{attribute 'qualified_only'}
{attribute 'strict'}
{attribute 'to_string'}
TYPE E_GridTypeSelection :
(
  Default             := 0,  // Default deformation based on cam points
  None                := 1,  // No deformation calculated all dx/dy=0
  Test_AllDxFactor    := 2,  // Dx constant for all = factor
  Test_AllDyFactor    := 3,  // Dy constant for all = factor
  Test_DyColFactor    := 4,  // Dy = col * factor (changes by column)
  Test_DxColFactor    := 5,  // Dx = col * factor (changes by column)
  Test_Dx_Row1OnlyFactor := 6   // dx factor only on row1 (test BOF)
) UINT := Default ;
END_TYPE

(* stored: Version 1.1.0.1, ProductVersion 3.1.4024.11
   EnumerationTextList E_GridTypeSelection: Id {b8f70bd9-6e05-42da-800f-ecab1d25db0a} *)
